PROGRAM S1_01_Motion_6
VAR
	HMI_Motion: FB_HMI_Control;
	Motion: FB_Motion2way;

	tMessageOffset: UINT;
	tNumMessagesPerRow: UINT;
	
	
	MyAdvanceInterlock: BOOL;
	MyReturnInterlock: BOOL;
	
	MyAutoAdvanceCondition: BOOL;
	MyAutoReturnCondition: BOOL;
	testword: WORD;
	myAdvancePrompt: BOOL;
	myReturnPrompt: BOOL;
	advancedSensor: BOOL;
	returnedSensor: BOOL;
	AdvanceCoil: BOOL;
	ReturnCoil: BOOL;
	tWaitMsgXICAdv: BOOL;
	tWaitMsgXICRet: BOOL;
	FB_SimMotion: FB_SimMotion;
	robToMarker: FB_RobotMotion;
	robToNowhere: FB_RobotMotion;
END_VAR

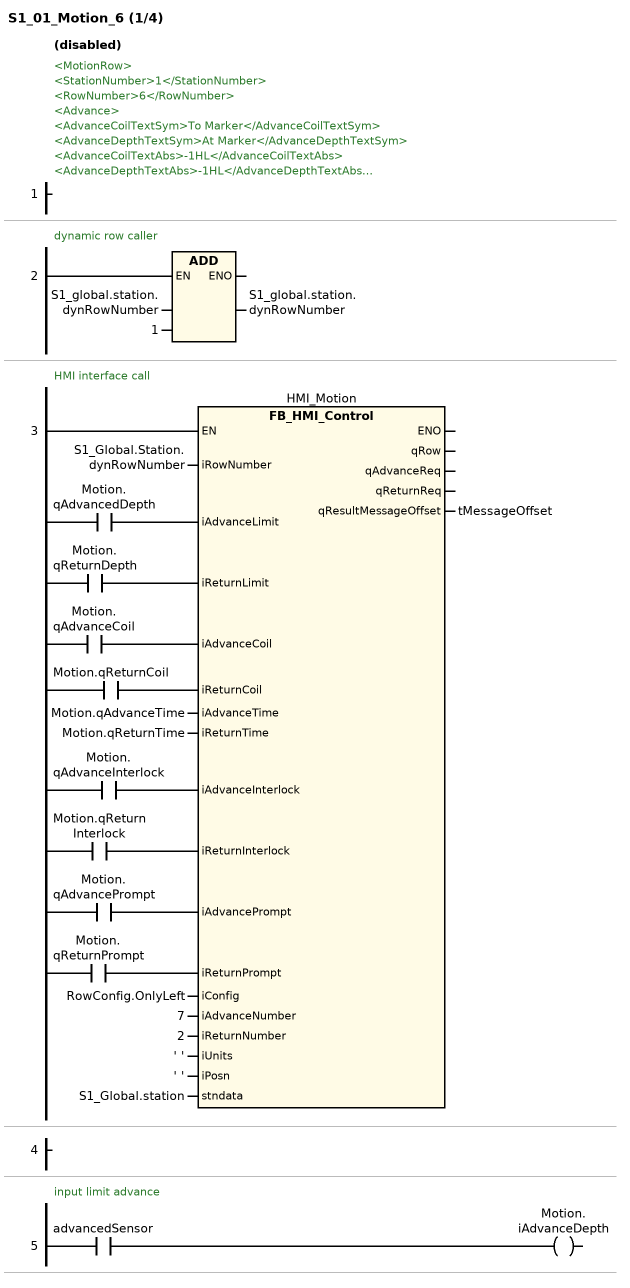
// NETWORK 1 (disabled)
// <MotionRow>
// <StationNumber>1</StationNumber>
// <RowNumber>6</RowNumber>
//   <Advance>
//     <AdvanceCoilTextSym>To Marker</AdvanceCoilTextSym>
//     <AdvanceDepthTextSym>At Marker</AdvanceDepthTextSym>
//     <AdvanceCoilTextAbs>-1HL</AdvanceCoilTextAbs>
//     <AdvanceDepthTextAbs>-1HL</AdvanceDepthTextAbs>
//     <ManSeq>7</ManSeq>
//   </Advance>
//   <Return>
//     <ReturnCoilTextSym>none</ReturnCoilTextSym>
//     <ReturnDepthTextSym>none</ReturnDepthTextSym>
//     <ReturnCoilTextAbs>none</ReturnCoilTextAbs>
//     <ReturnDepthTextAbs>none</ReturnDepthTextAbs>
//    <ManSeq>2</ManSeq>
//   </Return>
//   <Motion>
//     <NameSym>Robot</NameSym>
//     <NameAbs>-1HL</NameAbs>
//   </Motion>
// </MotionRow>

// NETWORK 2
// dynamic row caller
S1_global.station.dynRowNumber := S1_global.station.dynRowNumber + 1;

// NETWORK 3
// HMI interface call
HMI_Motion(
    iRowNumber := S1_Global.Station.dynRowNumber,
    iAdvanceLimit := Motion.qAdvancedDepth,
    iReturnLimit := Motion.qReturnDepth,
    iAdvanceCoil := Motion.qAdvanceCoil,
    iReturnCoil := Motion.qReturnCoil,
    iAdvanceTime := Motion.qAdvanceTime,
    iReturnTime := Motion.qReturnTime,
    iAdvanceInterlock := Motion.qAdvanceInterlock,
    iReturnInterlock := Motion.qReturnInterlock,
    iAdvancePrompt := Motion.qAdvancePrompt,
    iReturnPrompt := Motion.qReturnPrompt,
    iConfig := RowConfig.OnlyLeft,
    iAdvanceNumber := 7,
    iReturnNumber := 2,
    iUnits := ' ',
    iPosn := ' ',
    stndata := S1_Global.station,
    qResultMessageOffset => tMessageOffset); // FB_HMI_Control

// NETWORK 4

// NETWORK 5
// input limit advance
Motion.iAdvanceDepth := advancedSensor;

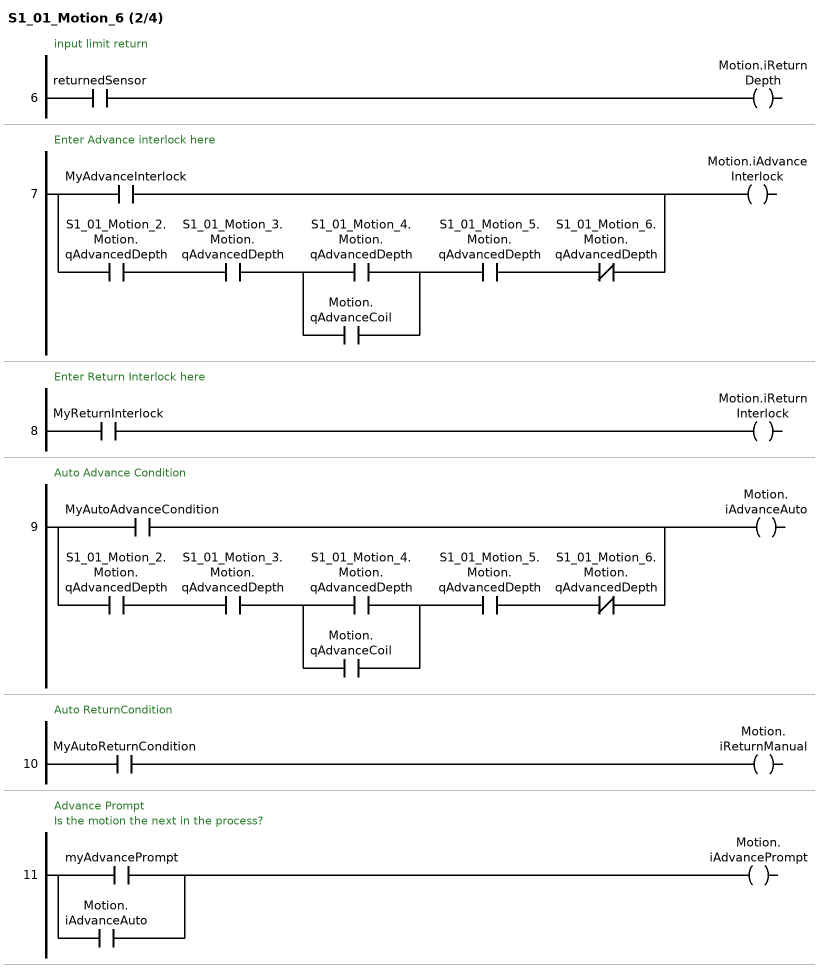
// NETWORK 6
// input limit return
Motion.iReturnDepth := returnedSensor;

// NETWORK 7
// Enter Advance interlock here
Motion.iAdvanceInterlock := MyAdvanceInterlock OR S1_01_Motion_2.Motion.qAdvancedDepth AND S1_01_Motion_3.Motion.qAdvancedDepth AND (S1_01_Motion_4.Motion.qAdvancedDepth OR Motion.qAdvanceCoil) AND S1_01_Motion_5.Motion.qAdvancedDepth AND NOT S1_01_Motion_6.Motion.qAdvancedDepth;

// NETWORK 8
// Enter Return Interlock here
Motion.iReturnInterlock := MyReturnInterlock;

// NETWORK 9
// Auto Advance Condition
Motion.iAdvanceAuto := MyAutoAdvanceCondition OR S1_01_Motion_2.Motion.qAdvancedDepth AND S1_01_Motion_3.Motion.qAdvancedDepth AND (S1_01_Motion_4.Motion.qAdvancedDepth OR Motion.qAdvanceCoil) AND S1_01_Motion_5.Motion.qAdvancedDepth AND NOT S1_01_Motion_6.Motion.qAdvancedDepth;

// NETWORK 10
// Auto ReturnCondition
Motion.iReturnManual := MyAutoReturnCondition;

// NETWORK 11
// Advance Prompt
// Is the motion the next in the process?
Motion.iAdvancePrompt := myAdvancePrompt OR Motion.iAdvanceAuto;

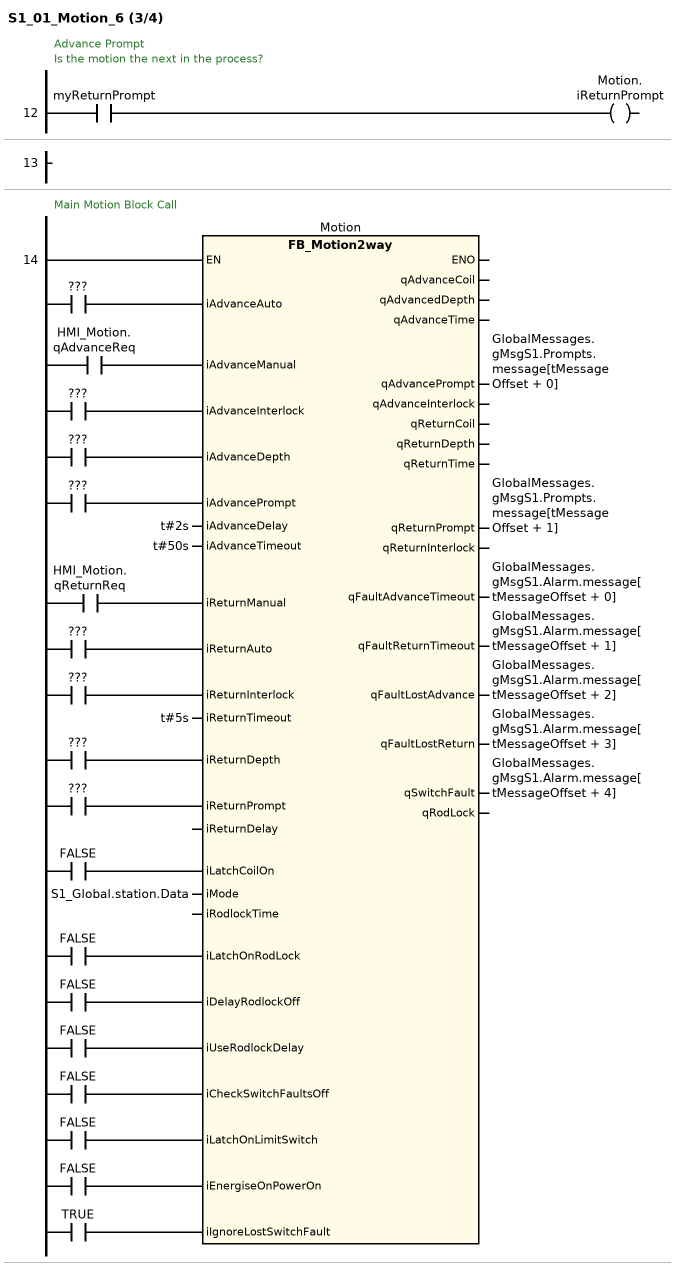
// NETWORK 12
// Advance Prompt
// Is the motion the next in the process?
Motion.iReturnPrompt := myReturnPrompt;

// NETWORK 13

// NETWORK 14
// Main Motion Block Call
Motion(
    iAdvanceManual := HMI_Motion.qAdvanceReq,
    iAdvanceDelay := t#2s,
    iAdvanceTimeout := t#50s,
    iReturnManual := HMI_Motion.qReturnReq,
    iReturnTimeout := t#5s,
    iLatchCoilOn := FALSE,
    iMode := S1_Global.station.Data,
    iLatchOnRodLock := FALSE,
    iDelayRodlockOff := FALSE,
    iUseRodlockDelay := FALSE,
    iCheckSwitchFaultsOff := FALSE,
    iLatchOnLimitSwitch := FALSE,
    iEnergiseOnPowerOn := FALSE,
    iIgnoreLostSwitchFault := TRUE,
    qAdvancePrompt => GlobalMessages.gMsgS1.Prompts.message[tMessageOffset + 0],
    qReturnPrompt => GlobalMessages.gMsgS1.Prompts.message[tMessageOffset + 1],
    qFaultAdvanceTimeout => GlobalMessages.gMsgS1.Alarm.message[tMessageOffset + 0],
    qFaultReturnTimeout => GlobalMessages.gMsgS1.Alarm.message[tMessageOffset + 1],
    qFaultLostAdvance => GlobalMessages.gMsgS1.Alarm.message[tMessageOffset + 2],
    qFaultLostReturn => GlobalMessages.gMsgS1.Alarm.message[tMessageOffset + 3],
    qSwitchFault => GlobalMessages.gMsgS1.Alarm.message[tMessageOffset + 4]); // FB_Motion2way

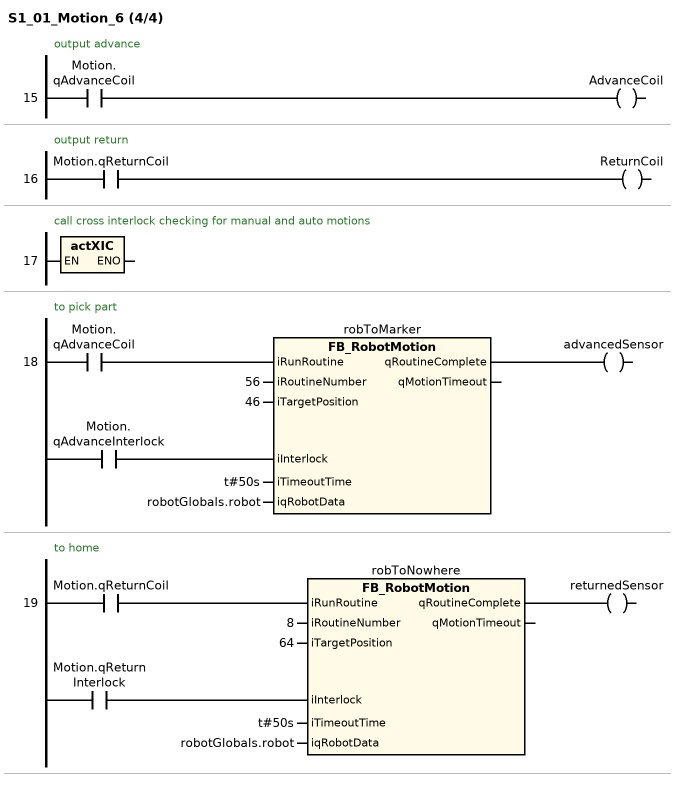
// NETWORK 15
// output advance
AdvanceCoil := Motion.qAdvanceCoil;

// NETWORK 16
// output return
ReturnCoil := Motion.qReturnCoil;

// NETWORK 17
// call cross interlock checking for manual and auto motions
actXIC();

// NETWORK 18
// to pick part
robToMarker(
    iRunRoutine := Motion.qAdvanceCoil,
    iRoutineNumber := 56,
    iTargetPosition := 46,
    iInterlock := Motion.qAdvanceInterlock,
    iTimeoutTime := t#50s,
    iqRobotData := robotGlobals.robot); // FB_RobotMotion
advancedSensor := robToMarker.qRoutineComplete;

// NETWORK 19
// to home
robToNowhere(
    iRunRoutine := Motion.qReturnCoil,
    iRoutineNumber := 8,
    iTargetPosition := 64,
    iInterlock := Motion.qReturnInterlock,
    iTimeoutTime := t#50s,
    iqRobotData := robotGlobals.robot); // FB_RobotMotion
returnedSensor := robToNowhere.qRoutineComplete;

ACTION actXIC:
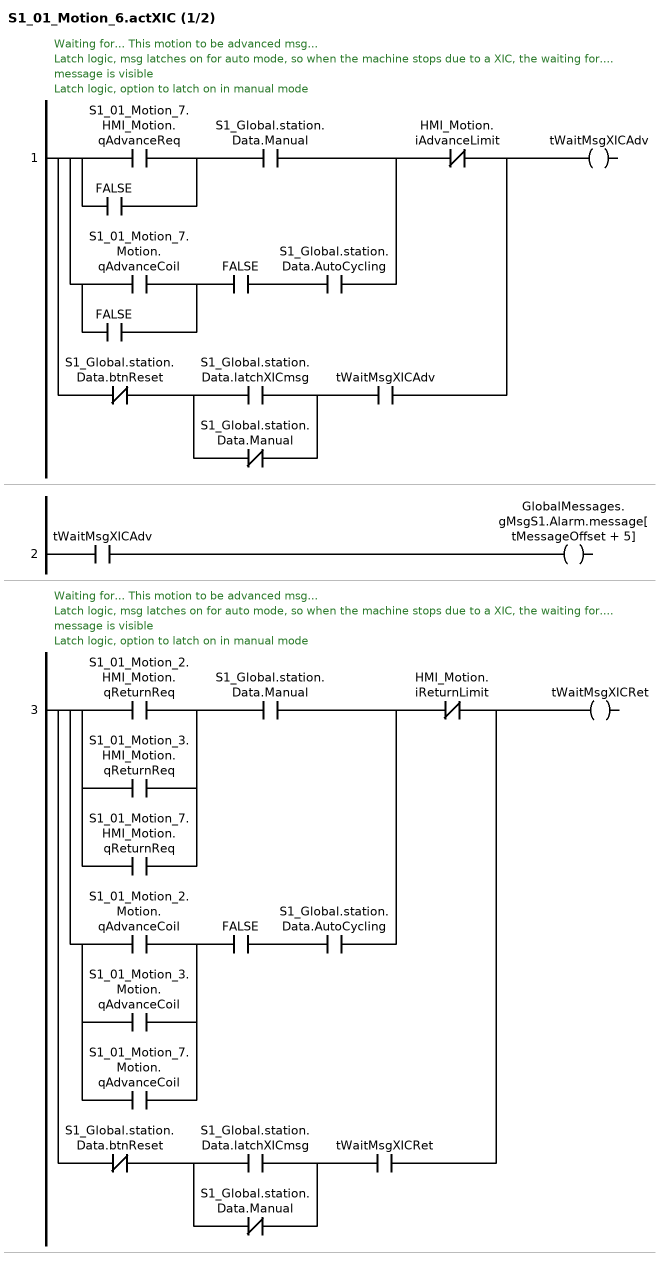
// NETWORK 1
// Waiting for... This motion to be advanced msg...
// Latch logic, msg latches on for auto mode, so when the machine stops due to a XIC, the waiting for.... message is visible
// Latch logic, option to latch on in manual mode
tWaitMsgXICAdv := ((S1_01_Motion_7.HMI_Motion.qAdvanceReq OR FALSE) AND S1_Global.station.Data.Manual OR (S1_01_Motion_7.Motion.qAdvanceCoil OR FALSE) AND FALSE AND S1_Global.station.Data.AutoCycling) AND NOT HMI_Motion.iAdvanceLimit OR NOT S1_Global.station.Data.btnReset AND (S1_Global.station.Data.latchXICmsg OR NOT S1_Global.station.Data.Manual) AND tWaitMsgXICAdv;

// NETWORK 2
GlobalMessages.gMsgS1.Alarm.message[tMessageOffset + 5] := tWaitMsgXICAdv;

// NETWORK 3
// Waiting for... This motion to be advanced msg...
// Latch logic, msg latches on for auto mode, so when the machine stops due to a XIC, the waiting for.... message is visible
// Latch logic, option to latch on in manual mode
tWaitMsgXICRet := ((S1_01_Motion_2.HMI_Motion.qReturnReq OR S1_01_Motion_3.HMI_Motion.qReturnReq OR S1_01_Motion_7.HMI_Motion.qReturnReq) AND S1_Global.station.Data.Manual OR (S1_01_Motion_2.Motion.qAdvanceCoil OR S1_01_Motion_3.Motion.qAdvanceCoil OR S1_01_Motion_7.Motion.qAdvanceCoil) AND FALSE AND S1_Global.station.Data.AutoCycling) AND NOT HMI_Motion.iReturnLimit OR NOT S1_Global.station.Data.btnReset AND (S1_Global.station.Data.latchXICmsg OR NOT S1_Global.station.Data.Manual) AND tWaitMsgXICRet;

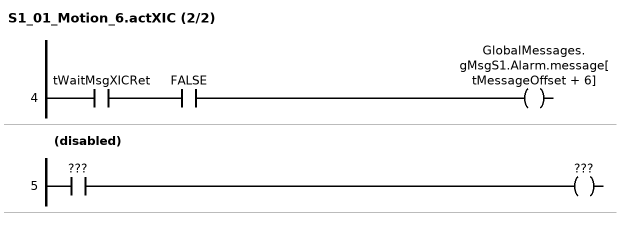
// NETWORK 4
GlobalMessages.gMsgS1.Alarm.message[tMessageOffset + 6] := tWaitMsgXICRet AND FALSE;

// NETWORK 5 (disabled)
// ??? := ???;
END_ACTION

END_PROGRAM

(* stored: Version 1.1.0.1, ProductVersion 3.1.4024.11
   POU S1_01_Motion_6: Id {5940c15b-76bb-456b-ac87-f823fd5b20e2}, SpecialFunc None
   Action actXIC: Id {c9149871-782b-0029-30c0-572ef7783b48} *)
